(* IEC 61131-3 sources: CS_4_Aufzugsteuerung/src/Stations/CP112/Steuerung/Class/clsEnableDrive, 1 file *)

(* ---- clsEnableDrive.st ---- *)
(*!
<Class
	Name               = "clsEnableDrive"
	Revision           = "0.0"
	RealtimeTask       = "false"
	CyclicTask         = "true"
	DefCyclictime      = "1 ms"
	BackgroundTask     = "false"
	Sigmatek           = "false"
	OSInterface        = "false"
	HighPriority       = "false"
	Automatic          = "false"
	UpdateMode         = "Prescan"
	SharedCommandTable = "true"
	Objectsize         = "(284,120)">
	<Channels>
		<Server Name="ClassSvr" Visualized="false" Initialize="false" WriteProtected="true" Retentive="false"/>
		<Client Name="cIn1" Required="true" Internal="false"/>
		<Client Name="cOut1" Required="true" Internal="false"/>
		<Client Name="cOut2" Required="true" Internal="false"/>
		<Client Name="cOut3" Required="true" Internal="false"/>
		<Client Name="cOut4" Required="true" Internal="false"/>
	</Channels>
</Class>
*)
clsEnableDrive : CLASS
  //Servers:
	ClassSvr 	: SvrChCmd_DINT;
  //Clients:
	cIn1 	: CltCh_DINT;
	cOut1 	: CltCh_DINT;
	cOut2 	: CltCh_DINT;
	cOut3 	: CltCh_DINT;
	cOut4 	: CltCh_DINT;
  //Variables:
  //Functions:

	FUNCTION VIRTUAL GLOBAL CyWork
		VAR_INPUT
			EAX 	: UDINT;
		END_VAR
		VAR_OUTPUT
			state (EAX) 	: UDINT;
		END_VAR;
  //Tables:
	FUNCTION @STD
		VAR_OUTPUT
			ret_code	: CONFSTATES;
		END_VAR;
	FUNCTION GLOBAL TAB @CT_;
END_CLASS;

FUNCTION VIRTUAL GLOBAL clsEnableDrive::CyWork
	VAR_INPUT
		EAX 	: UDINT;
	END_VAR
	VAR_OUTPUT
		state (EAX) 	: UDINT;
	END_VAR

  cIn1 := cIn1.Read ();

  cOut1 := cOut2 := cOut3 := cOut4 := cIn1;
  cOut1.Write (cOut1);
  cOut2.Write (cOut2);
  cOut3.Write (cOut3);
  cOut4.Write (cOut4);

	state := READY;

END_FUNCTION
